/// MODULE INTERFACE INPUT AND OUTPUT 
TYPE DUT_MODULE_INTERFACE :
STRUCT
	///Information that the module reads
	Input: DUT_MODULE_INTERFACE_INPUT;
	///Information that the module write
	Output: DUT_MODULE_INTERFACE_OUTPUT;
END_STRUCT
END_TYPE

(* stored: Version 1.1.0.1, ProductVersion 3.1.0.25
   DUT DUT_MODULE_INTERFACE: Id {eeb4175f-f5ee-4644-806e-62eb9e62eee0} *)
